{attribute addProperty BoxType "EL6080-0000-0016"}
{attribute addProperty Id "StatusAT %I*Status_77B8DE54000InputsEMPTY_STRUCTURE000ControlAT %Q*Control_AB2F34C6000OutputsEMPTY_STRUCTURE000WcStateAT %I*WcState_F855686C1620InfoDataAT %I*InfoData_BC63D37F80100"}
{attribute addProperty CRC "2407072411"}
{attribute addProperty SizeInBites "96"}
{attribute addProperty SizeInBytes "12"}
TYPE EL6080_49EF2FC4 :
STRUCT
	{attribute addProperty Name "Status"}
	Status : Status_77B8DE54;
	{attribute addProperty Name "Inputs"}
	Inputs : EMPTY_STRUCTURE;
	{attribute addProperty Name "Control"}
	Control : Control_AB2F34C6;
	{attribute addProperty Name "Outputs"}
	Outputs : EMPTY_STRUCTURE;
	{attribute addProperty Name "WcState"}
	WcState : WcState_F855686C;
	{attribute addProperty Name "InfoData"}
	InfoData : InfoData_BC63D37F;
END_STRUCT
END_TYPE

(* stored: Version 1.2.0.0, ProductVersion 3.1.4024.9
   DUT EL6080_49EF2FC4: Id {f96bc4db-1daa-44b3-a7c9-2fd02c9ae2d9} *)
